{attribute addProperty BoxType "EK1122-0000-0018"}
{attribute addProperty Id "Beckhoff_EL99xxsub_EK1100EK1100_179A0949162"}
{attribute addProperty CRC "1229738181"}
{attribute addProperty SizeInBites "16"}
{attribute addProperty SizeInBytes "2"}
TYPE Beckhoff_EL99xxEK1122_494C50C5 EXTENDS EK1122_179A0949 :
STRUCT
	{attribute addProperty Name "Beckhoff_EL99xxsub_EK1100"}
	Beckhoff_EL99xxsub_EK1100 : EK1100_179A0949;
END_STRUCT
END_TYPE

(* stored: Version 1.2.0.0, ProductVersion 3.1.4024.9
   DUT Beckhoff_EL99xxEK1122_494C50C5: Id {e953c209-9673-4e1b-b366-0618803f1c6d} *)
